{attribute addProperty BoxType "EL2521-0124-0016"}
{attribute addProperty Id "Enable_PLSAT %Q*BOOL811OutputAT %Q*BOOL814Switch_on_valueAT %Q*UINT16217Switch_off_valueAT %Q*UINT16218"}
{attribute addProperty CRC "313489322"}
{attribute addProperty SizeInBites "48"}
{attribute addProperty SizeInBytes "6"}
TYPE PLS_Control_compact_12AF77AA :
STRUCT
	{attribute addProperty Name "Enable_PLS"}
	Enable_PLS AT %Q* : BOOL;
	{attribute addProperty Name "Output"}
	Output AT %Q* : BOOL;
	{attribute addProperty Name "Switch_on_value"}
	Switch_on_value AT %Q* : UINT;
	{attribute addProperty Name "Switch_off_value"}
	Switch_off_value AT %Q* : UINT;
END_STRUCT
END_TYPE

(* stored: Version 1.2.0.0, ProductVersion 3.1.4024.9
   DUT PLS_Control_compact_12AF77AA: Id {99b82030-9d30-431a-92d9-07126dc2d054} *)
